// TIA Portal V15.1 export
// export: Created 2026-01-15T16:29:43.7391028Z, ExportSetting WithDefaults, WithReadOnly, DisplayName Totally Integrated Automation Portal, DisplayVersion V15.1 Update 8, DisplayName TIA Portal Openness, DisplayVersion V15.1 Update 8, DisplayName STEP 7 Professional, DisplayVersion V15.1 Update 8, DisplayName WinCC Advanced, DisplayVersion V15.1 Update 8
DATA_BLOCK "7.4.ADD6"   // DB719
{ S7_Optimized_Access := 'TRUE' }
VERSION : 0.1
// stored: AutoNumber true, CodeModifiedDate 2026-01-15T16:25:55.9362535Z, CompileDate 2026-01-15T16:25:55.9409287Z, CreationDate 2026-01-15T16:22:49.8270549Z, DBAccessibleFromOPCUA true, DownloadWithoutReinit false, InstanceOfName 7.WEIGHT_PROCESS, InstanceOfNumber 7, InstanceOfType FB, InterfaceModifiedDate 2024-08-06T09:13:34.3012657Z, IsConsistent true, IsKnowHowProtected false, IsRetainMemResEnabled false, MemoryReserve 100, ModifiedDate 2026-01-15T16:25:55.9362535Z, ParameterModified 2024-08-06T08:53:48.4792275Z, StructureModified 2024-08-06T09:13:34.3012657Z, UDAEnableTagReadback false
"7.WEIGHT_PROCESS"
   // VAR_INPUT
   //    AUT : Bool;
   //    MAN1 : Bool;
   //    MAN2 : Bool;
   //    LOGIC : Bool;
   //    FAU : Bool;
   //    FU_IN : Bool;
   //    X_CLOCK : Bool;
   //    EMTY_IN : Bool;
   //    XNC_MAN : Bool;
   //    XNC_AUT : Bool;
   //    BU_TRU : Bool;
   //    SV_IN : Real;
   //    W_IN : Real;
   //    W_RTD : Real;
   //    W_TR : Real;
   //    W_DU : Real;
   //    T_ON : Real;
   //    T_OFF : Real;
   //    T_DL : Real;
   //    SMT : Real;
   //    KL_Bu_Tru : Real;
   // END_VAR
   // VAR_OUTPUT
   //    MAC_OUT : Real;
   //    PV_OUT : Real;
   //    PVA_OUT : Real;
   //    PVM_OUT : Real;
   //    FU_OUT : Bool;
   //    EM_OUT : Bool;
   //    W_OVER : Real;
   //    Q_OUT1 : Bool;
   //    Q_OUT2 : Bool;
   //    OVER : Bool;
   //    STA_RUN : Bool;
   // END_VAR
   // VAR RETAIN
   //    FU { ExternalAccessible := 'False'; ExternalVisible := 'False'; ExternalWritable := 'False'} : Bool;
   //    EM { ExternalAccessible := 'False'; ExternalVisible := 'False'; ExternalWritable := 'False'} : Bool;
   //    "CAN DU" { ExternalAccessible := 'False'; ExternalVisible := 'False'; ExternalWritable := 'False'} : Real;
   //    PVA { ExternalAccessible := 'False'; ExternalVisible := 'False'; ExternalWritable := 'False'} : Real;
   //    PVM { ExternalAccessible := 'False'; ExternalVisible := 'False'; ExternalWritable := 'False'} : Real;
   //    TOFF { ExternalAccessible := 'False'; ExternalVisible := 'False'; ExternalWritable := 'False'} : Real;
   //    TON { ExternalAccessible := 'False'; ExternalVisible := 'False'; ExternalWritable := 'False'} : Real;
   //    T_DLFULL { ExternalAccessible := 'False'; ExternalVisible := 'False'; ExternalWritable := 'False'} : Real;
   //    "T_DLT/T" { ExternalAccessible := 'False'; ExternalVisible := 'False'; ExternalWritable := 'False'} : Real;
   //    KL_BU : Real;
   //    CLK_DLE { ExternalAccessible := 'False'; ExternalVisible := 'False'; ExternalWritable := 'False'} : Bool;
   //    CLK_DLF { ExternalAccessible := 'False'; ExternalVisible := 'False'; ExternalWritable := 'False'} : Bool;
   //    "CLK_DLT/T" { ExternalAccessible := 'False'; ExternalVisible := 'False'; ExternalWritable := 'False'} : Bool;
   //    CLK_TT { ExternalAccessible := 'False'; ExternalVisible := 'False'; ExternalWritable := 'False'} : Bool;
   //    "TEMP_T/T" { ExternalAccessible := 'False'; ExternalVisible := 'False'; ExternalWritable := 'False'} : Bool;
   //    "RUN_T/T" { ExternalAccessible := 'False'; ExternalVisible := 'False'; ExternalWritable := 'False'} : Bool;
   // END_VAR
   // VAR
   //    RUN_MAN : Bool;
   //    RUN_AUT : Bool;
   //    "CUA_T/T" : Bool;
   //    P_OUT1 : Bool;
   //    P_OUT2 : Bool;
   //    P_EMTY : Bool;
   //    P_FU : Bool;
   // END_VAR
BEGIN
END_DATA_BLOCK
